SYSTEM ASM_MVL (* Assembly System Model+View+HMI *)
  (* Standard: 61499-1; Classification: Simulation; ApplicationDomain: Assembly; Type: Dual Stroke Cylinder *)
  (* Version 0.0, 2004-09-25, JHC, Rockwell Automation, Adapted from ASM_MVL using simpler components. *)
  DEVICE MODEL : FRAME_DEVICE
    RESOURCE CLOCK : EMB_RES
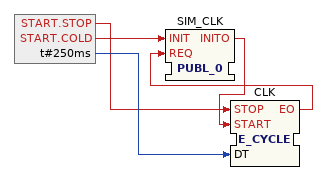
      FBS
        CLK : E_CYCLE;
        SIM_CLK : PUBL_0;
      END_FBS
      EVENT_CONNECTIONS
        START.STOP TO CLK.STOP;
        START.COLD TO SIM_CLK.INIT;
        SIM_CLK.INITO TO CLK.START;
        CLK.EO TO SIM_CLK.REQ;
      END_CONNECTIONS
      DATA_CONNECTIONS
        t#250ms TO CLK.DT;
      END_CONNECTIONS
    END_RESOURCE
    RESOURCE TRANSPORT_MDL : PANEL_RESOURCE
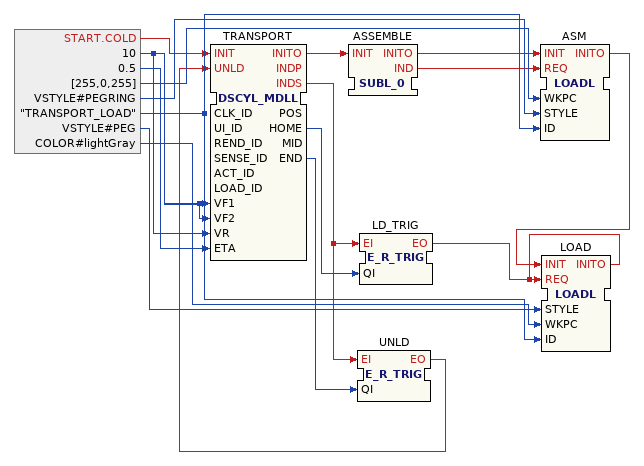
      FBS
        TRANSPORT : DSCYL_MDLL;
        UNLD : E_R_TRIG;
        ASM : LOADL;
        LD_TRIG : E_R_TRIG;
        ASSEMBLE : SUBL_0;
        LOAD : LOADL;
      END_FBS
      EVENT_CONNECTIONS
        TRANSPORT.INDS TO UNLD.EI;
        TRANSPORT.INDS TO LD_TRIG.EI;
        START.COLD TO TRANSPORT.INIT;
        TRANSPORT.INITO TO ASSEMBLE.INIT;
        ASSEMBLE.INITO TO ASM.INIT;
        ASSEMBLE.IND TO ASM.REQ;
        UNLD.EO TO TRANSPORT.UNLD;
        ASM.INITO TO LOAD.INIT;
        LOAD.INITO TO LOAD.REQ;
        LD_TRIG.EO TO LOAD.REQ;
      END_CONNECTIONS
      DATA_CONNECTIONS
        TRANSPORT.END TO UNLD.QI;
        TRANSPORT.HOME TO LD_TRIG.QI;
        10 TO TRANSPORT.VF1;
        10 TO TRANSPORT.VF2;
        10 TO TRANSPORT.VR;
        0.5 TO TRANSPORT.ETA;
        [255,0,255] TO ASM.WKPC;
        VSTYLE#PEGRING TO ASM.STYLE;
        "TRANSPORT_LOAD" TO ASM.ID;
        VSTYLE#PEG TO LOAD.STYLE;
        COLOR#lightGray TO LOAD.WKPC;
        "TRANSPORT_LOAD" TO LOAD.ID;
      END_CONNECTIONS
    END_RESOURCE
    RESOURCE PRESS_MDL : PANEL_RESOURCE
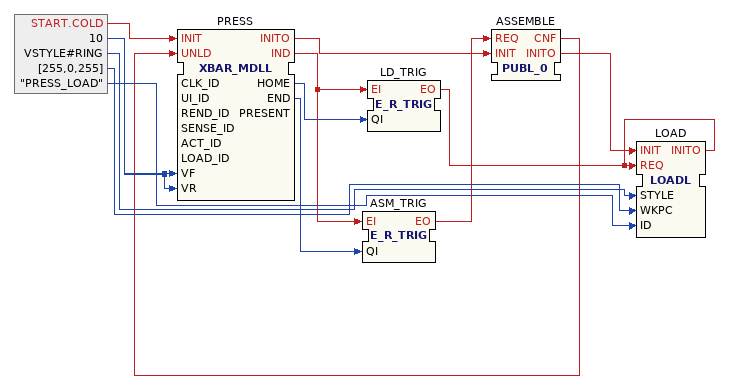
      FBS
        PRESS : XBAR_MDLL;
        ASM_TRIG : E_R_TRIG; (* Gate for assembly event *)
        ASSEMBLE : PUBL_0;
        LD_TRIG : E_R_TRIG;
        LOAD : LOADL;
      END_FBS
      EVENT_CONNECTIONS
        ASM_TRIG.EO TO ASSEMBLE.REQ;
        START.COLD TO PRESS.INIT;
        PRESS.IND TO LD_TRIG.EI;
        PRESS.IND TO ASM_TRIG.EI;
        PRESS.INITO TO ASSEMBLE.INIT;
        ASSEMBLE.CNF TO PRESS.UNLD;
        ASSEMBLE.INITO TO LOAD.INIT;
        LD_TRIG.EO TO LOAD.REQ;
        LOAD.INITO TO LOAD.REQ;
      END_CONNECTIONS
      DATA_CONNECTIONS
        PRESS.END TO ASM_TRIG.QI;
        10 TO PRESS.VF;
        10 TO PRESS.VR;
        PRESS.HOME TO LD_TRIG.QI;
        VSTYLE#RING TO LOAD.STYLE;
        [255,0,255] TO LOAD.WKPC;
        "PRESS_LOAD" TO LOAD.ID;
      END_CONNECTIONS
    END_RESOURCE
    RESOURCE ASSEMBLY : VIEW_PANEL
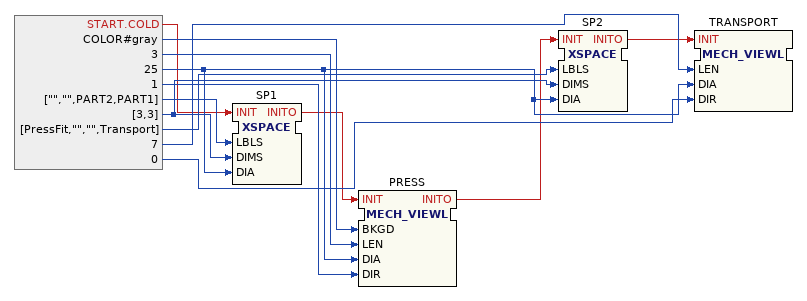
      FBS
        SP1 : XSPACE;
        PRESS : MECH_VIEWL; (* Vertical press element *)
        SP2 : XSPACE;
        TRANSPORT : MECH_VIEWL; (* Dual-Cylinder Transport Mechanism *)
      END_FBS
      EVENT_CONNECTIONS
        START.COLD TO SP1.INIT;
        SP1.INITO TO PRESS.INIT;
        PRESS.INITO TO SP2.INIT;
        SP2.INITO TO TRANSPORT.INIT;
      END_CONNECTIONS
      DATA_CONNECTIONS
        COLOR#gray TO PRESS.BKGD;
        3 TO PRESS.LEN;
        25 TO PRESS.DIA;
        1 TO PRESS.DIR;
        ["","",PART2,PART1] TO SP1.LBLS;
        [3,3] TO SP1.DIMS;
        25 TO SP1.DIA;
        [PressFit,"","",Transport] TO SP2.LBLS;
        [3,3] TO SP2.DIMS;
        25 TO SP2.DIA;
        7 TO TRANSPORT.LEN;
        25 TO TRANSPORT.DIA;
        0 TO TRANSPORT.DIR;
      END_CONNECTIONS
    END_RESOURCE
    DATA_CONNECTIONS
      0 TO ASSEMBLY.TRACE;
      25 TO ASSEMBLY.DIA;
      [7,5] TO ASSEMBLY.SIZE;
      0 TO ASSEMBLY.VERTICAL;
    END_CONNECTIONS
  END_DEVICE
  DEVICE HMI : FRAME_DEVICE
    RESOURCE TRANSPORT_SENSORS : PANEL_RESOURCE
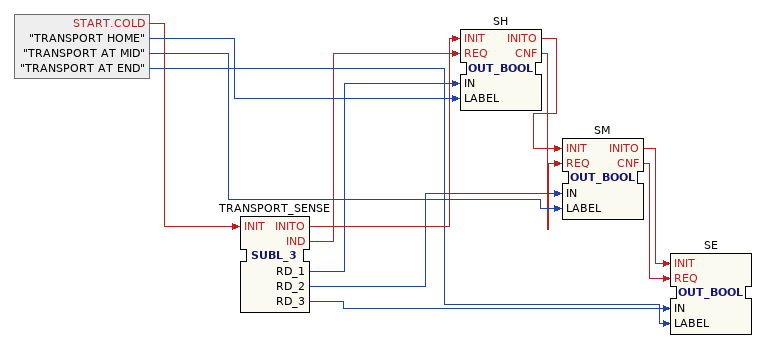
      FBS
        TRANSPORT_SENSE : SUBL_3;
        SH : OUT_BOOL;
        SM : OUT_BOOL;
        SE : OUT_BOOL;
      END_FBS
      EVENT_CONNECTIONS
        START.COLD TO TRANSPORT_SENSE.INIT;
        TRANSPORT_SENSE.INITO TO SH.INIT;
        SH.INITO TO SM.INIT;
        SM.INITO TO SE.INIT;
        TRANSPORT_SENSE.IND TO SH.REQ;
        SH.CNF TO SM.REQ;
        SM.CNF TO SE.REQ;
      END_CONNECTIONS
      DATA_CONNECTIONS
        TRANSPORT_SENSE.RD_1 TO SH.IN;
        TRANSPORT_SENSE.RD_2 TO SM.IN;
        TRANSPORT_SENSE.RD_3 TO SE.IN;
        "TRANSPORT HOME" TO SH.LABEL;
        "TRANSPORT AT MID" TO SM.LABEL;
        "TRANSPORT AT END" TO SE.LABEL;
      END_CONNECTIONS
    END_RESOURCE
    RESOURCE TRANSPORT_ACTUATORS : PANEL_RESOURCE
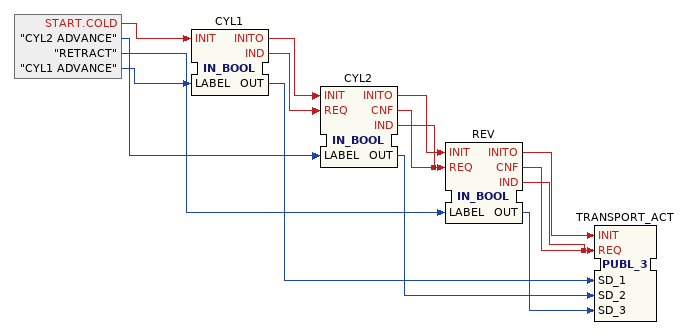
      FBS
        CYL1 : IN_BOOL;
        CYL2 : IN_BOOL;
        REV : IN_BOOL;
        TRANSPORT_ACT : PUBL_3;
      END_FBS
      EVENT_CONNECTIONS
        START.COLD TO CYL1.INIT;
        CYL1.INITO TO CYL2.INIT;
        CYL2.INITO TO REV.INIT;
        REV.INITO TO TRANSPORT_ACT.INIT;
        CYL1.IND TO CYL2.REQ;
        CYL2.CNF TO REV.REQ;
        CYL2.IND TO REV.REQ;
        REV.CNF TO TRANSPORT_ACT.REQ;
        REV.IND TO TRANSPORT_ACT.REQ;
      END_CONNECTIONS
      DATA_CONNECTIONS
        CYL1.OUT TO TRANSPORT_ACT.SD_1;
        CYL2.OUT TO TRANSPORT_ACT.SD_2;
        REV.OUT TO TRANSPORT_ACT.SD_3;
        "CYL2 ADVANCE" TO CYL2.LABEL;
        "RETRACT" TO REV.LABEL;
        "CYL1 ADVANCE" TO CYL1.LABEL;
      END_CONNECTIONS
    END_RESOURCE
    RESOURCE PRESS_SENSORS : PANEL_RESOURCE
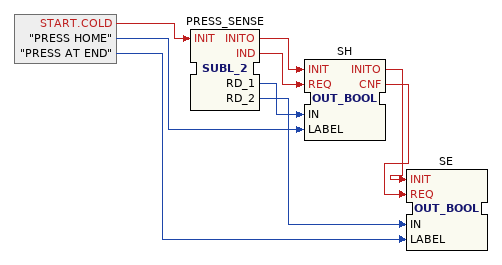
      FBS
        PRESS_SENSE : SUBL_2;
        SH : OUT_BOOL;
        SE : OUT_BOOL;
      END_FBS
      EVENT_CONNECTIONS
        START.COLD TO PRESS_SENSE.INIT;
        PRESS_SENSE.INITO TO SH.INIT;
        SH.INITO TO SE.INIT;
        PRESS_SENSE.IND TO SH.REQ;
        SH.CNF TO SE.REQ;
      END_CONNECTIONS
      DATA_CONNECTIONS
        PRESS_SENSE.RD_1 TO SH.IN;
        PRESS_SENSE.RD_2 TO SE.IN;
        "PRESS HOME" TO SH.LABEL;
        "PRESS AT END" TO SE.LABEL;
      END_CONNECTIONS
    END_RESOURCE
    RESOURCE PRESS_ACTUATORS : PANEL_RESOURCE
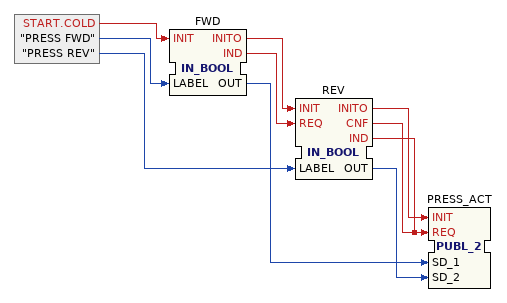
      FBS
        FWD : IN_BOOL;
        REV : IN_BOOL;
        PRESS_ACT : PUBL_2;
      END_FBS
      EVENT_CONNECTIONS
        START.COLD TO FWD.INIT;
        FWD.INITO TO REV.INIT;
        REV.INITO TO PRESS_ACT.INIT;
        FWD.IND TO REV.REQ;
        REV.CNF TO PRESS_ACT.REQ;
        REV.IND TO PRESS_ACT.REQ;
      END_CONNECTIONS
      DATA_CONNECTIONS
        FWD.OUT TO PRESS_ACT.SD_1;
        REV.OUT TO PRESS_ACT.SD_2;
        "PRESS FWD" TO FWD.LABEL;
        "PRESS REV" TO REV.LABEL;
      END_CONNECTIONS
    END_RESOURCE
    DATA_CONNECTIONS
      3 TO TRANSPORT_SENSORS.ROWS;
      1 TO TRANSPORT_SENSORS.COLS;
      3 TO TRANSPORT_ACTUATORS.ROWS;
      1 TO TRANSPORT_ACTUATORS.COLS;
      3 TO PRESS_SENSORS.ROWS;
      1 TO PRESS_SENSORS.COLS;
      3 TO PRESS_ACTUATORS.ROWS;
      1 TO PRESS_ACTUATORS.COLS;
    END_CONNECTIONS
  END_DEVICE
  DATA_CONNECTIONS (* parameter values *)
    [460,100,185,150] TO MODEL.BOUNDS;
    [460,100,185,150] TO MODEL.BOUNDS;
    [100,100,360,150] TO HMI.BOUNDS;
    [2,2] TO HMI.GRID;
  END_CONNECTIONS
END_SYSTEM
